Yaskawa INFORM job: B-4-08279-80-0-L.JBI

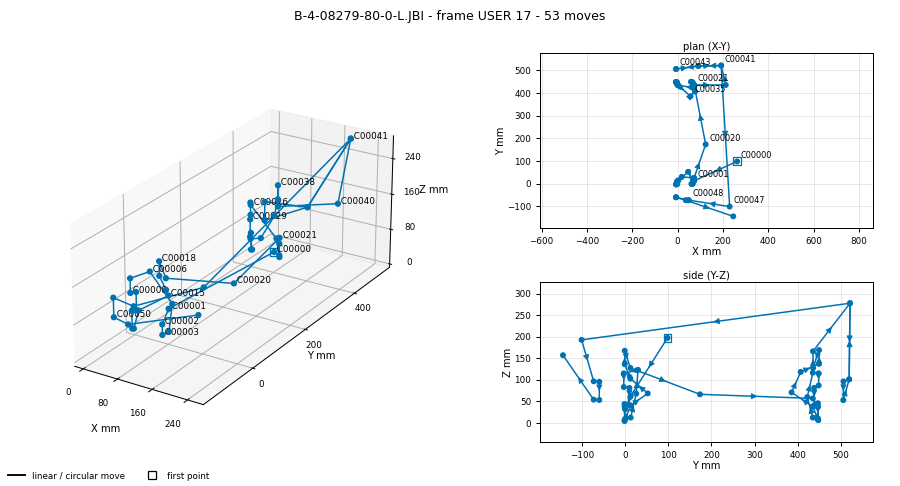
[picture p0: tool path of B-4-08279-80-0-L.JBI in frame USER 17, 53 of 53 moves have a stored position in this frame; points joined in program order, loops and branches not executed]
/JOB
//NAME B-4-08279-80-0-L
///FOLDERNAME PART_420-08279-80
//POS
///NPOS 53,0,53,0,0,0
///USER 17
///TOOL 4
///POSTYPE USER
///RECTAN
///RCONF 1,0,0,0,0,0,0,0,0,0,0,0,0,0,0,0,0,0,0,0,0,0,0,0
C00000=262.619,98.241,197.316,-96.7907,26.0612,130.3907
C00001=73.206,12.887,62.532,-108.1130,33.6440,124.7280
C00002=66.350,-0.100,32.103,-108.1108,33.6415,124.7296
C00003=66.144,-0.064,8.818,-108.1102,33.6417,124.7294
C00004=73.207,12.886,12.496,-108.1130,33.6440,124.7280
C00005=73.209,25.753,68.034,-108.1130,33.6440,124.7280
C00006=18.285,29.861,123.023,-105.1660,8.3780,132.7380
C00007=-6.287,-3.209,115.149,-105.4078,23.2277,133.7821
C00008=-6.480,-3.150,83.385,-105.4099,23.2272,133.7808
C00009=-1.744,9.833,81.413,-106.8820,26.9670,127.1640
C00010=-1.744,9.833,41.151,-106.8820,26.9670,127.1640
C00011=-5.062,-1.610,44.144,-106.0157,27.8877,132.1438
C00012=-5.041,-1.269,4.809,-123.5777,18.2473,128.8974
C00013=-1.290,-1.274,5.760,-123.5776,18.2478,128.8971
C00014=1.309,12.886,40.637,-115.9500,15.0640,123.8880
C00015=46.568,52.366,68.637,-115.9500,15.0640,123.8880
C00016=68.126,12.203,102.713,-51.9240,65.1860,170.4170
C00017=61.579,-0.942,136.189,-52.1440,65.1479,170.2046
C00018=61.935,-0.974,167.433,-52.1454,65.1479,170.2039
C00019=68.127,12.203,127.579,-51.9240,65.1860,170.4170
C00020=123.702,173.377,66.504,-51.9240,65.1860,170.4170
C00021=73.207,435.046,56.988,108.1130,33.6440,-124.7280
C00022=65.666,446.732,37.273,108.1143,33.6435,-124.7266
C00023=65.725,446.752,10.542,108.1139,33.6425,-124.7265
C00024=73.207,435.046,12.497,108.1130,33.6440,-124.7280
C00025=73.208,422.239,60.087,108.1130,33.6440,-124.7280
C00026=1.310,435.046,116.590,106.4700,24.0930,-128.1180
C00027=-7.724,448.586,115.133,105.5302,25.0980,-133.5412
C00028=-7.135,448.600,87.014,105.5281,25.0989,-133.5401
C00029=-1.744,438.100,81.414,106.4700,24.0930,-128.1180
C00030=-1.744,438.100,41.152,106.4700,24.0930,-128.1180
C00031=-5.366,447.020,45.781,105.2449,25.3652,-135.1521
C00032=-5.213,447.521,6.771,115.5919,16.8005,-135.0662
C00033=-2.606,447.501,7.423,115.5969,16.7960,-135.0671
C00034=1.310,435.046,37.856,114.8060,13.4990,-125.4170
C00035=56.824,385.802,71.014,114.8060,13.4990,-125.4170
C00036=76.829,406.941,118.422,51.9240,65.1860,-170.4170
C00037=59.646,449.436,137.153,51.9366,65.1831,-170.4089
C00038=59.660,449.447,169.020,51.9328,65.1825,-170.4118
C00039=68.127,435.729,127.579,51.9240,65.1860,-170.4170
C00040=212.373,435.445,166.233,51.9240,65.1860,-170.4170
C00041=191.994,521.318,277.669,-64.9580,52.3036,155.2869
C00042=91.520,519.266,101.171,-160.3299,74.1577,66.0982
C00043=-6.736,506.042,96.398,-160.3218,74.1573,66.1082
C00044=-7.072,505.666,53.064,-160.3258,74.1576,66.1034
C00045=91.520,519.266,101.171,-160.3299,74.1577,66.0982
C00046=191.994,521.318,277.669,-64.9580,52.3036,155.2869
C00047=229.653,-100.956,192.660,69.2460,43.0800,-149.5110
C00048=49.647,-72.877,96.659,69.2460,43.0800,-149.5110
C00049=-7.409,-59.907,95.583,69.2459,43.0780,-149.5114
C00050=-7.232,-59.895,53.304,69.2452,43.0802,-149.5116
C00051=35.736,-72.877,54.138,69.2460,43.0800,-149.5110
C00052=245.487,-144.122,157.206,69.2470,43.0790,-149.5110
///TOOL 0
///POSTYPE ANGLE
///ANGLE
EC00000=15.0000
///TOOL 4
EC00001=15.0000
///TOOL 0
EC00002=15.0000
EC00003=15.0000
///TOOL 4
EC00004=15.0000
EC00005=15.0000
EC00006=15.0000
///TOOL 0
EC00007=15.0000
EC00008=15.0000
///TOOL 4
EC00009=15.0000
EC00010=15.0000
///TOOL 0
EC00011=15.0000
EC00012=14.9994
EC00013=14.9994
///TOOL 4
EC00014=15.0000
EC00015=15.0000
EC00016=15.0000
///TOOL 0
EC00017=15.0000
EC00018=15.0000
///TOOL 4
EC00019=15.0000
EC00020=15.0000
EC00021=15.0000
///TOOL 0
EC00022=15.0000
EC00023=15.0000
///TOOL 4
EC00024=15.0000
EC00025=15.0000
EC00026=15.0000
///TOOL 0
EC00027=15.0000
EC00028=15.0000
///TOOL 4
EC00029=15.0000
EC00030=15.0000
///TOOL 0
EC00031=15.0000
EC00032=15.0000
EC00033=15.0000
///TOOL 4
EC00034=15.0000
EC00035=15.0000
EC00036=15.0000
///TOOL 0
EC00037=15.0000
EC00038=15.0000
///TOOL 4
EC00039=15.0000
EC00040=15.0000
///TOOL 0
EC00041=15.0000
EC00042=15.0000
EC00043=15.0000
EC00044=15.0000
EC00045=15.0000
EC00046=15.0000
///TOOL 4
EC00047=15.0000
EC00048=15.0000
///TOOL 0
EC00049=15.0000
EC00050=15.0000
///TOOL 4
EC00051=15.0000
EC00052=15.0000
//INST
///DATE 2021/10/29 11:36
///ATTR SC,RW,RJ
////FRAME USER 17
///GROUP1 RB1
///GROUP2 ST3
NOP
'Path Start: PP56
MOVJ C00000 VJ=100.00  +MOVJ EC00000
SMOVL C00001 V=1250.0  +MOVJ EC00001
SMOVL C00002 V=300.0  +MOVJ EC00002
ARCON ASF#(953)
SMOVL C00003 V=8.5  +MOVJ EC00003
ARCOF AEF#(953)
SMOVL C00004 V=1250.0  +MOVJ EC00004
SMOVL C00005 V=1250.0  +MOVJ EC00005
'Path End
'Path Start: PP54
SMOVL C00006 V=1250.0  +MOVJ EC00006
SMOVL C00007 V=300.0  +MOVJ EC00007
ARCON ASF#(952)
SMOVL C00008 V=6.3  +MOVJ EC00008
ARCOF AEF#(954)
SMOVL C00009 V=300.0  +MOVJ EC00009
SMOVL C00010 V=300.0  +MOVJ EC00010
SMOVL C00011 V=300.0  +MOVJ EC00011
ARCON ASF#(952)
SMOVL C00012 V=6.3  +MOVJ EC00012
SMOVL C00013 V=6.3  +MOVJ EC00013
ARCOF AEF#(954)
SMOVL C00014 V=1250.0  +MOVJ EC00014
SMOVL C00015 V=1250.0  +MOVJ EC00015
'Path End
'Path Start: Path_5
SMOVL C00016 V=1250.0  +MOVJ EC00016
SMOVL C00017 V=1250.0  +MOVJ EC00017
ARCON ASF#(951)
SMOVL C00018 V=8.5  +MOVJ EC00018
ARCOF AEF#(951)
SMOVL C00019 V=1250.0  +MOVJ EC00019
SMOVL C00020 V=1250.0  +MOVJ EC00020
'Path End
'Path Start: PP55
SMOVL C00021 V=1250.0  +MOVJ EC00021
SMOVL C00022 V=300.0  +MOVJ EC00022
ARCON ASF#(953)
SMOVL C00023 V=8.5  +MOVJ EC00023
ARCOF AEF#(953)
SMOVL C00024 V=1250.0  +MOVJ EC00024
SMOVL C00025 V=1250.0  +MOVJ EC00025
'Path End
'Path Start: PP58
SMOVL C00026 V=1250.0  +MOVJ EC00026
SMOVL C00027 V=300.0  +MOVJ EC00027
ARCON ASF#(952)
SMOVL C00028 V=6.3  +MOVJ EC00028
ARCOF AEF#(954)
SMOVL C00029 V=300.0  +MOVJ EC00029
SMOVL C00030 V=300.0  +MOVJ EC00030
SMOVL C00031 V=300.0  +MOVJ EC00031
ARCON ASF#(952)
SMOVL C00032 V=6.3  +MOVJ EC00032
SMOVL C00033 V=6.3  +MOVJ EC00033
ARCOF AEF#(954)
SMOVL C00034 V=1250.0  +MOVJ EC00034
SMOVL C00035 V=1250.0  +MOVJ EC00035
'Path End
'Path Start: Path_4
SMOVL C00036 V=1250.0  +MOVJ EC00036
SMOVL C00037 V=1250.0  +MOVJ EC00037
ARCON ASF#(951)
SMOVL C00038 V=8.5  +MOVJ EC00038
ARCOF AEF#(951)
SMOVL C00039 V=1250.0  +MOVJ EC00039
SMOVL C00040 V=1250.0  +MOVJ EC00040
'Path End
'Path Start: PP57
SMOVL C00041 V=1250.0  +MOVJ EC00041
SMOVL C00042 V=1250.0  +MOVJ EC00042
SMOVL C00043 V=300.0  +MOVJ EC00043
ARCON ASF#(953)
SMOVL C00044 V=8.5  +MOVJ EC00044
ARCOF AEF#(953)
SMOVL C00045 V=1250.0  +MOVJ EC00045
SMOVL C00046 V=1250.0  +MOVJ EC00046
'Path End
'Path Start: PP53
SMOVL C00047 V=1250.0  +MOVJ EC00047
SMOVL C00048 V=1250.0  +MOVJ EC00048
SMOVL C00049 V=300.0  +MOVJ EC00049
ARCON ASF#(953)
SMOVL C00050 V=8.5  +MOVJ EC00050
ARCOF AEF#(953)
SMOVL C00051 V=1250.0  +MOVJ EC00051
SMOVL C00052 V=1250.0  +MOVJ EC00052
'Path End
END
